// TIA Portal V20 export
FUNCTION_BLOCK "FSFB_Main_Safety_RTG1"   // FB1, F_FBD
   VAR
      ESTOP : ESTOP1;
   END_VAR
BEGIN

REGION Network 1
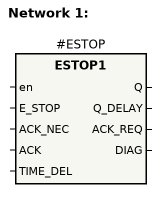
   #ESTOP();   // ESTOP1
END_REGION
END_FUNCTION_BLOCK
